FUNCTION F_AddPadding : STRING
VAR_INPUT
	nNumber:		INT;
	nSize:			UINT;
END_VAR
VAR
	sTemp: STRING;
END_VAR

sTemp := INT_TO_STRING(nNumber);

WHILE LEN(sTemp) < nSize DO
	sTemp := CONCAT('0',sTemp);
END_WHILE

F_AddPadding := sTemp;

END_FUNCTION

(* stored: Version 1.1.0.1, ProductVersion 3.1.4024.15
   POU F_AddPadding: Id {719dc483-a24f-4f03-975b-5d06842ab86a}, SpecialFunc None *)
